// TwinCAT 3 PLC project PLC_1
// ProgramVersion: 3.1.4024.0
// libraries:
//   Tc2_Math, * (Beckhoff Automation GmbH)
//   Tc2_MC2, * (Beckhoff Automation GmbH)
//   Tc2_Standard, * (Beckhoff Automation GmbH)
//   Tc2_System, * (Beckhoff Automation GmbH)
//   Tc3_Module, * (Beckhoff Automation GmbH)
// project tree:
//   / PlcTask.TcTTO
//   POUs/ KinematicControl.TcPOU, MAIN.TcPOU, MasterAxisControl.TcPOU, SlaveAxisControl.TcPOU
// real-time tasks:
//   TASK PlcTask: cycle T#10ms, priority 20, ADS port 350
// motion (NC):
//   TASK NC-Task 1 SAF: cycle T#2ms, priority 4, ADS port 501
//   TASK NC-Task 1 SVB: cycle T#10ms, priority 8, ADS port 511
//   AXIS Master (id 3)
//     OtherSettings: AllowMotionCmdToSlave=true
//     encoder EncType=1
//     drive DrvType=5
//       Analog: TorqueSetpointScale=10, ScaleFactorActTorque=0.1
//     controller CtrType=1
//       CtrPara: PriorControlFactor=1
//         Observer: BandWidth=20
//   AXIS Slave 1 (id 4)
//     OtherSettings: AllowMotionCmdToSlave=true
//     encoder EncType=1
//     drive DrvType=5
//       Analog: TorqueSetpointScale=10, ScaleFactorActTorque=0.1
//     controller CtrType=1
//       CtrPara: PriorControlFactor=1
//         Observer: BandWidth=20
//   AXIS Slave 2 (id 5)
//     OtherSettings: AllowMotionCmdToSlave=true
//     encoder EncType=1
//     drive DrvType=5
//       Analog: TorqueSetpointScale=10, ScaleFactorActTorque=0.1
//     controller CtrType=1
//       CtrPara: PriorControlFactor=1
//         Observer: BandWidth=20
//   AXIS Slave 3 (id 6)
//     OtherSettings: AllowMotionCmdToSlave=true
//     encoder EncType=1
//     drive DrvType=5
//       Analog: TorqueSetpointScale=10, ScaleFactorActTorque=0.1
//     controller CtrType=1
//       CtrPara: PriorControlFactor=1
//         Observer: BandWidth=20
//   AXIS Master Axis (id 1)
//     General: UnitName=°, UnitFlags=#x00000004
//     OtherSettings: AllowMotionCmdToSlave=true
//     encoder EncType=1
//       EncPara: EncMode=3
//     drive DrvType=5
//       Analog: TorqueSetpointScale=10, ScaleFactorActTorque=0.1
//       TimeComp: TaskDelayCycles=1
//     controller CtrType=1
//       CtrPara: PriorControlFactor=1
//         Observer: BandWidth=20
//   AXIS Slave Axis (id 2)
//     General: UnitName=°, UnitFlags=#x00000004
//     OtherSettings: AllowMotionCmdToSlave=true
//     encoder EncType=1
//     drive DrvType=5
//       Analog: TorqueSetpointScale=10, ScaleFactorActTorque=0.1
//       TimeComp: TaskDelayCycles=1
//     controller CtrType=1
//       CtrPara: PriorControlFactor=1
//         Observer: BandWidth=20
// variable links:
//   PLC 1/PLC 1 Instance <-> NC-Task 1 SAF/Axes/Master Axis
//     PlcTask Inputs/MAIN.MasterAxis._Axis.NcToPlc <-> Outputs/ToPlc
//     PlcTask Outputs/MAIN.MasterAxis._Axis.PlcToNc <-> Inputs/FromPlc
//   PLC 1/PLC 1 Instance <-> NC-Task 1 SAF/Axes/Slave Axis
//     PlcTask Inputs/MAIN.SlaveAxis._Axis.NcToPlc <-> Outputs/ToPlc
//     PlcTask Outputs/MAIN.SlaveAxis._Axis.PlcToNc <-> Inputs/FromPlc

CONFIGURATION PLC_1
    RESOURCE PLC ON TwinCAT3
        TASK PlcTask(INTERVAL := T#10ms, PRIORITY := 20);
        PROGRAM MAIN WITH PlcTask : MAIN;
    END_RESOURCE
END_CONFIGURATION

// ---- POUs/MAIN.TcPOU
PROGRAM MAIN
VAR
	
	MasterAxis		: MasterAxisControl;
	SlaveAxis		: SlaveAxisControl;
	Length			: LREAL := 200;
	Width			: LREAL := 40;
	Size			: LREAL := 80;
	xStart			: LREAL := 800;
	yStart			: LREAL := 400;
	State			: BYTE;
	
	Kinematic		: KinematicControl;
	
END_VAR

MasterAxis.CyclicUpdate();
SlaveAxis.CyclicUpdate();

MasterAxis.LengthOfShaft		 	:= Length;
MasterAxis.WidthOfShaft 			:= Width;
MasterAxis.AxisSize 				:= Size;
MasterAxis.XCoord 					:= xStart;
MasterAxis.YCoord 					:= yStart;

SlaveAxis.LengthOfShaft 			:= 150;
SlaveAxis.WidthOfShaft 				:= 60;
SlaveAxis.PreviousWidthOfShaft 		:= MasterAxis.WidthOfShaft;
SlaveAxis.PreviousAnglePosition 	:= MasterAxis.AnglePosition;
SlaveAxis.PreviousLengthOfShaft 	:= MasterAxis.LengthOfShaft;

SlaveAxis.PreviousXCoordGlobal 		:= MasterAxis.XCoord;
SlaveAxis.PreviousYCoordGlobal 		:= MasterAxis.YCoord;
SlaveAxis.PreviousXCoordRelative	:= MasterAxis.XCoord;
SlaveAxis.PreviousYCoordRelative	:= MasterAxis.YCoord;

CASE State OF
	
	0:
		IF MasterAxis.PowerOn() AND_THEN SlaveAxis.PowerOn() THEN
			State := 1;
		END_IF
		
	1:
		MasterAxis.MoveRelative(Position := 360, Velocity := 10);
	
END_CASE




Kinematic.CyclicUpdate();

END_PROGRAM

// ---- POUs/MasterAxisControl.TcPOU
FUNCTION_BLOCK MasterAxisControl
VAR
	
	_Axis			: AXIS_REF;
	
	_AnglePosition	: LREAL;
	_LengthOfShaft	: LREAL;
	_WidthOfShaft	: LREAL;
	_AxisSize		: LREAL;
	_xCoordRelative	: LREAL;
	_yCoordRelative	: LREAL;
	_LocalState		: BYTE;
	
	_Enable			: MC_Power;
	_Reset			: MC_Reset;
	_MovePosAbs		: MC_MoveAbsolute;
	_MovePosRel		: MC_MoveRelative;	
	_ReadStatus		: MC_ReadStatus;
	
END_VAR

PROPERTY AnglePosition : LREAL
GET
AnglePosition := _AnglePosition;
END_GET
SET
END_SET
END_PROPERTY

PROPERTY AxisSize : LREAL
GET
AxisSize := _AxisSize;
END_GET
SET
IF AxisSize < 0 THEN
	_AxisSize := 0;
ELSE
	_AxisSize := AxisSize;
END_IF
END_SET
END_PROPERTY

METHOD CyclicUpdate : BOOL
VAR_INPUT
END_VAR
_Enable(Axis := _Axis);
_Reset(Axis := _Axis);
_ReadStatus(Axis := _Axis);
_MovePosAbs(Axis := _Axis);
_MovePosRel(Axis := _Axis);

_AnglePosition := _Axis.NcToPlc.ModuloActPos;
END_METHOD

PROPERTY LengthOfShaft : LREAL
GET
LengthOfShaft := _LengthOfShaft;
END_GET
SET
IF LengthOfShaft < 0 THEN
	_LengthOfShaft := 0;
ELSE
	_LengthOfShaft := LengthOfShaft;
END_IF
END_SET
END_PROPERTY

METHOD MoveRelative : BOOL
VAR_INPUT
	Position	: LREAL;
	Velocity	: LREAL;
END_VAR
_MovePosRel(Axis := _Axis);
_MovePosRel.Distance := Position;
_MovePosRel.Velocity := Velocity;
_MovePosRel.Execute := TRUE;
IF _MovePosRel.Done THEN
	_MovePosRel.Execute := FALSE;
	MoveRelative := TRUE;
ELSIF _MovePosRel.Error THEN
	_MovePosRel.Execute := FALSE;
	MoveRelative := FALSE;
END_IF
END_METHOD

METHOD PowerOn : BOOL
VAR_INPUT
END_VAR
_Enable(Axis := _Axis);
_Enable.Enable := TRUE;
_Enable.Enable_Negative := TRUE;
_Enable.Enable_Positive := TRUE;
_Enable.Override := 100;
IF _Enable.Status THEN
	PowerOn := TRUE;
END_IF
END_METHOD

PROPERTY WidthOfShaft : LREAL
GET
WidthOfShaft := _WidthOfShaft;
END_GET
SET
IF WidthOfShaft < 0 THEN
	_WidthOfShaft := 0;
ELSE
	_WidthOfShaft := WidthOfShaft;
END_IF
END_SET
END_PROPERTY

PROPERTY XCoord : LREAL
GET
XCoord := _xCoordRelative;
END_GET
SET
_xCoordRelative := XCoord;
END_SET
END_PROPERTY

PROPERTY YCoord : LREAL
GET
YCoord := _yCoordRelative;
END_GET
SET
_yCoordRelative := YCoord;
END_SET
END_PROPERTY

END_FUNCTION_BLOCK

// ---- POUs/SlaveAxisControl.TcPOU
FUNCTION_BLOCK SlaveAxisControl EXTENDS MasterAxisControl
VAR
	
	_PreviousAnglePosition		: LREAL;
	_PreviousLengthOfShaft		: LREAL;
	_PreviousWidthOfShaft		: LREAL;
	
	_xCoordPreviousRelative		: LREAL;
	_yCoordPreviousRelative		: LREAL;
	_xCoordPreviousGlobal		: LREAL;
	_yCoordPreviousGlobal		: LREAL;
	_xCoordGlobal				: LREAL;
	_yCoordGlobal				: LREAL;
	
	_SlaveOrderInChain			: LREAL;
	
END_VAR

METHOD CyclicUpdate : BOOL
VAR_INPUT
END_VAR
_Enable(Axis := _Axis);
_Reset(Axis := _Axis);
_ReadStatus(Axis := _Axis);
_MovePosAbs(Axis := _Axis);
_MovePosRel(Axis := _Axis);

_xCoordRelative := _PreviousLengthOfShaft * COS(_PreviousAnglePosition * Pi / 180);
_yCoordRelative := _PreviousLengthOfShaft * SIN(_PreviousAnglePosition * Pi / 180);

_xCoordGlobal := _xCoordRelative + _xCoordPreviousGlobal;
_yCoordGlobal := _yCoordRelative + _yCoordPreviousGlobal;
END_METHOD

PROPERTY PreviousAnglePosition : LREAL
GET
PreviousAnglePosition := _PreviousAnglePosition;
END_GET
SET
_PreviousAnglePosition := PreviousAnglePosition;
END_SET
END_PROPERTY

PROPERTY PreviousLengthOfShaft : LREAL
GET
PreviousLengthOfShaft := _PreviousLengthOfShaft;
END_GET
SET
_PreviousLengthOfShaft := PreviousLengthOfShaft;
END_SET
END_PROPERTY

PROPERTY PreviousWidthOfShaft : LREAL
GET
PreviousWidthOfShaft := _PreviousWidthOfShaft;
END_GET
SET
_PreviousWidthOfShaft := PreviousWidthOfShaft;
END_SET
END_PROPERTY

PROPERTY PreviousXCoordGlobal : LREAL
GET
PreviousXCoordGlobal := _xCoordPreviousGlobal;
END_GET
SET
_xCoordPreviousGlobal := PreviousXCoordGlobal;
END_SET
END_PROPERTY

PROPERTY PreviousXCoordRelative : LREAL
GET
PreviousXCoordRelative := _xCoordPreviousRelative;
END_GET
SET
_xCoordPreviousRelative := PreviousXCoordRelative;
END_SET
END_PROPERTY

PROPERTY PreviousYCoordGlobal : LREAL
GET
PreviousYCoordGlobal := _yCoordPreviousGlobal;
END_GET
SET
_yCoordPreviousGlobal := PreviousYCoordGlobal;
END_SET
END_PROPERTY

PROPERTY PreviousYCoordRelative : LREAL
GET
PreviousYCoordRelative := _yCoordPreviousRelative;
END_GET
SET
_yCoordPreviousRelative := PreviousYCoordRelative;
END_SET
END_PROPERTY

PROPERTY SlaveOrderInChain : LREAL
GET
SlaveOrderInChain := _SlaveOrderInChain;
END_GET
SET
IF SlaveOrderInChain < 1 THEN
	_SlaveOrderInChain := 1;
ELSE
	_SlaveOrderInChain := SlaveOrderInChain;
END_IF
END_SET
END_PROPERTY

END_FUNCTION_BLOCK

// ---- POUs/KinematicControl.TcPOU
FUNCTION_BLOCK KinematicControl
VAR
	
	_Master				: MasterAxisControl;
	_Slave				: ARRAY [1.._NumOfSlaves] OF SlaveAxisControl;
	
	_LocalState			: BYTE;
	_i					: BYTE;
	
END_VAR
VAR CONSTANT
	
	_NumOfSlaves		: BYTE := 3;

END_VAR

METHOD CyclicUpdate : BOOL
VAR_INPUT
END_VAR

// Update all axes
_Master.CyclicUpdate();
FOR _i := 1 TO _NumOfSlaves BY 1 DO
	_Slave[_i].CyclicUpdate();
END_FOR

_Slave[1].PreviousAnglePosition 	:= _Master.AnglePosition;
_Slave[1].PreviousLengthOfShaft 	:= _Master.LengthOfShaft;
_Slave[1].PreviousWidthOfShaft		:= _Master.WidthOfShaft;
_Slave[1].PreviousXCoordGlobal		:= _Master.XCoord;
_Slave[1].PreviousYCoordGlobal		:= _Master.YCoord;

IF _NumOfSlaves > 1 THEN
	FOR _i := 2 TO _NumOfSlaves BY 1 DO
		_Slave[_i].PreviousAnglePosition	:= _Slave[_i - 1].AnglePosition;
		_Slave[_i].PreviousLengthOfShaft 	:= _Slave[_i - 1].LengthOfShaft;
		_Slave[_i].PreviousWidthOfShaft		:= _Slave[_i - 1].WidthOfShaft;
		_Slave[_i].PreviousXCoordGlobal		:= _Slave[_i - 1].XCoord;
		_Slave[_i].PreviousYCoordGlobal		:= _Slave[_i - 1].YCoord;
	END_FOR	
END_IF
END_METHOD

END_FUNCTION_BLOCK
